(* IEC 61131-3 sources: DirIOHMI/src/Ar/DirIOHMI, 3 files *)

(* ---- DirIOHMI.typ ---- *)
(*
 * File: DirIOHMI.typ
 * Copyright (c) 2023 Loupe
 * https://loupe.team
 *
 * This file is part of DirIOHMI, licensed under the MIT License.
 *)

TYPE
	DirectoryMgr_HMI_typ : 	STRUCT
		Enable : BOOL;
		Main : DirectoryMgr_HMI_Main_typ;
		Pane : ARRAY[0..1]OF DirectoryMgr_HMI_Browser_typ;
		Progress : DirectoryMgr_HMI_Progress_typ;
		internal : DirectoryMgr_internal_typ;
	END_STRUCT;
	DirectoryMgr_HMI_Main_typ : 	STRUCT
		CopyLeftToRight : HMI_Button_typ;
		CopyRightToLeft : HMI_Button_typ;
		ExtensionList : ARRAY[0..9]OF STRING[260];
	END_STRUCT;
	DirectoryMgr_HMI_Browser_typ : 	STRUCT
		CreateDirectory : HMI_Button_typ;
		Delete : HMI_Button_typ;
		Rename : HMI_Button_typ;
		ToFile : HMI_Button_typ;
		ToDataObject : HMI_Button_typ;
		Browser : HMIFileBrowse;
		Progress : DirectoryMgr_HMI_Progress_typ;
		FileList : ARRAY[0..19]OF STRING[260];
		IgnoreErrors : USINT;
		ErrorString : STRING[DIOWRAP_STRLEN_ERROR];
	END_STRUCT;
	DirectoryMgr_HMI_Progress_typ : 	STRUCT
		StatusDP : UINT;
		Progress : UDINT;
	END_STRUCT;
	DirectoryMgr_internal_typ : 	STRUCT
		ErrorString : STRING[DIOWRAP_STRLEN_ERROR];
	END_STRUCT;
END_TYPE

(* ---- DirIOHMI.fun ---- *)
(*
 * File: DirIOHMI.fun
 * Copyright (c) 2023 Loupe
 * https://loupe.team
 *
 * This file is part of DirIOHMI, licensed under the MIT License.
 *)

FUNCTION DirIODualPane : BOOL (* *) (*$GROUP=User*)
	VAR_INPUT
		HMI : DirectoryMgr_HMI_typ;
	END_VAR
	VAR_IN_OUT
		t : DIOWrap_typ;
	END_VAR
END_FUNCTION

FUNCTION DirIOPane : BOOL (* *) (*$GROUP=User*)
	VAR_INPUT
		Pane : DirectoryMgr_HMI_Browser_typ;
	END_VAR
	VAR_IN_OUT
		t : DIOWrap_typ;
	END_VAR
END_FUNCTION

(* ---- DirIOHMI.var ---- *)
(*
 * File: DirIOHMI.var
 * Copyright (c) 2023 Loupe
 * https://loupe.team
 *
 * This file is part of DirIOHMI, licensed under the MIT License.
 *)
VAR CONSTANT
	DIOWRAP_DO_NAME_LEN : UINT := 260;
	DIOWRAP_DO_LIST_LEN : UINT := 20;
END_VAR
